{attribute addProperty BoxType "EK1100-0000-0018"}
{attribute addProperty Id "Beckhoff_AX86xxEK1122Beckhoff_AX86xxEK1122_9E61CBD75848731"}
{attribute addProperty CRC "507257289"}
{attribute addProperty SizeInBites "5848"}
{attribute addProperty SizeInBytes "731"}
TYPE Beckhoff_AX86xx_1E3C21C9 EXTENDS EK1100_179A0949 :
STRUCT
	{attribute addProperty Name "Beckhoff_AX86xxEK1122"}
	Beckhoff_AX86xxEK1122 : Beckhoff_AX86xxEK1122_9E61CBD7;
END_STRUCT
END_TYPE

(* stored: Version 1.2.0.0, ProductVersion 3.1.4024.9
   DUT Beckhoff_AX86xx_1E3C21C9: Id {6ac33f91-f04f-4049-8575-01cc28f693ec} *)
